TYPE 
  ST_SystemStatus_AR : ARRAY [0..C.uiNumIrrLinesForHMI_C] OF ST_SystemStatus;
END_TYPE

(* stored: Version 1.1.0.1, ProductVersion 3.1.4024.12
   DUT ST_SystemStatus_AR: Id {3e2a39c0-dca3-4c28-a8bc-86f57f9af2bd} *)
